TYPE ST_WallPermission :
STRUCT
    IsPermittedToEnter    : BOOL; //TRUE if permitted to enter the wall
    IsNotPermittedToEnter : BOOL; //TRUE if not permitted to enter
    IsNotPermittedToExit  : BOOL; //TRUE if not permitted to exit
END_STRUCT
END_TYPE

(* stored: Version 1.1.0.1, ProductVersion 3.1.4024.11
   DUT ST_WallPermission: Id {84903c25-5a8c-0968-2ec8-c223c497da2f} *)
